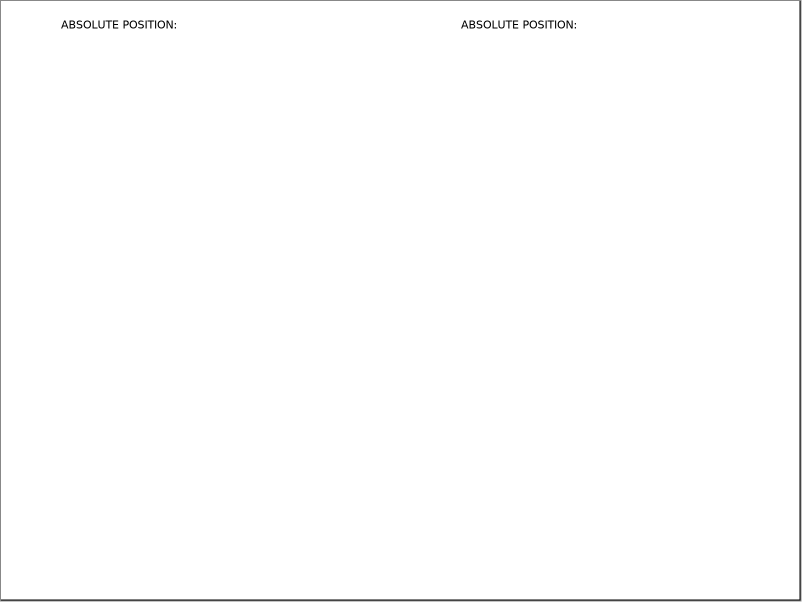
VISUALIZATION F39_Acceleration_Profile  // 802x602
    Rectangle (0,0 800x600)
    Label (10,10 170x30), "ABSOLUTE POSITION:"
    Label (410,10 170x30), "ABSOLUTE POSITION:"
END_VISUALIZATION

(* stored: Version 1.1.0.1, ProductVersion 3.1.4022.7
   Visu F39_Acceleration_Profile: Id {ee91234a-22c3-4b9f-97a7-5e6a94e05b9a} *)
